Universal Robots URScript: external_control.urscript

{{BEGIN_REPLACE}}

# HEADER_BEGIN

steptime = get_steptime()

textmsg("ExternalControl: steptime=", steptime)
MULT_jointstate = {{JOINT_STATE_REPLACE}}
MULT_time = {{TIME_REPLACE}}

STOPJ_ACCELERATION = 4.0

#Constants
SERVO_UNINITIALIZED = -1
SERVO_IDLE = 0
SERVO_RUNNING = 1

MODE_STOPPED = -2
MODE_UNINITIALIZED = -1
MODE_IDLE = 0
MODE_SERVOJ = 1
MODE_SPEEDJ = 2
MODE_FORWARD = 3
MODE_SPEEDL = 4
MODE_POSE = 5
MODE_SPLINE = 6

TRAJECTORY_MODE_RECEIVE = 1
TRAJECTORY_MODE_CANCEL = -1

TRAJECTORY_POINT_INTERPOLATION = 0
TRAJECTORY_SPLINE_INTERPOLATION = 1

TRAJECTORY_POINT_JOINT = 0
TRAJECTORY_POINT_CARTESIAN = 1
TRAJECTORY_DATA_DIMENSION = 7

TRAJECTORY_RESULT_SUCCESS = 0
TRAJECTORY_RESULT_CANCELED = 1
TRAJECTORY_RESULT_FAILURE = 2

CUBIC_SPLINES = 0
QUINTIC_SPLINES = 1

TRAJECTORY_SPLINE_DATA_DIMENSION = 3*6 + 2

#Global variables are also showed in the Teach pendants variable list
global cmd_servo_state = SERVO_UNINITIALIZED
global cmd_servo_qd = [0.0, 0.0, 0.0, 0.0, 0.0, 0.0]
global cmd_servo_q = get_actual_joint_positions()
global cmd_servo_q_last = get_actual_joint_positions()
global cmd_twist = [0.0, 0.0, 0.0, 0.0, 0.0, 0.0]
global extrapolate_count = 0
global extrapolate_max_count = 0
global control_mode = MODE_UNINITIALIZED
global trajectory_points_left = 0

def set_servo_setpoint(params_mult):
  cmd_servo_state = SERVO_RUNNING
  cmd_servo_q_last = cmd_servo_q
  cmd_servo_q = [params_mult[2] / MULT_jointstate, params_mult[3] / MULT_jointstate, params_mult[4] / MULT_jointstate, params_mult[5] / MULT_jointstate, params_mult[6] / MULT_jointstate, params_mult[7] / MULT_jointstate]
end

def extrapolate():
  diff = [cmd_servo_q[0] - cmd_servo_q_last[0], cmd_servo_q[1] - cmd_servo_q_last[1], cmd_servo_q[2] - cmd_servo_q_last[2], cmd_servo_q[3] - cmd_servo_q_last[3], cmd_servo_q[4] - cmd_servo_q_last[4], cmd_servo_q[5] - cmd_servo_q_last[5]]
  cmd_servo_q_last = cmd_servo_q
  cmd_servo_q = [cmd_servo_q[0] + diff[0], cmd_servo_q[1] + diff[1], cmd_servo_q[2] + diff[2], cmd_servo_q[3] + diff[3], cmd_servo_q[4] + diff[4], cmd_servo_q[5] + diff[5]]

  return cmd_servo_q
end

thread servoThread():
  textmsg("ExternalControl: Starting servo thread")
  state = SERVO_IDLE
  while control_mode == MODE_SERVOJ:
    enter_critical
    q = cmd_servo_q
    do_extrapolate = False
    if (cmd_servo_state == SERVO_IDLE):
      do_extrapolate = True
    end
    state = cmd_servo_state
    if cmd_servo_state > SERVO_UNINITIALIZED:
      cmd_servo_state = SERVO_IDLE
    end

    if do_extrapolate:
      extrapolate_count = extrapolate_count + 1
      if extrapolate_count > extrapolate_max_count:
        extrapolate_max_count = extrapolate_count
      end

      q = extrapolate()
      servoj(q, t=steptime, {{SERVO_J_REPLACE}})

    elif state == SERVO_RUNNING:
      extrapolate_count = 0
      servoj(q, t=steptime, {{SERVO_J_REPLACE}})
    else:
      extrapolate_count = 0
      sync()
    end
    exit_critical
  end
  textmsg("ExternalControl: servo thread ended")
  stopj(STOPJ_ACCELERATION)
end

# Helpers for speed control
def set_speed(params_mult):
  cmd_servo_qd = [params_mult[2] / MULT_jointstate, params_mult[3] / MULT_jointstate, params_mult[4] / MULT_jointstate, params_mult[5] / MULT_jointstate, params_mult[6] / MULT_jointstate, params_mult[7] / MULT_jointstate]
  control_mode = MODE_SPEEDJ
end

thread speedThread():
  textmsg("ExternalControl: Starting speed thread")
  while control_mode == MODE_SPEEDJ:
    qd = cmd_servo_qd
    speedj(qd, 40.0, steptime)
  end
  textmsg("ExternalControl: speedj thread ended")
  stopj(STOPJ_ACCELERATION)
end

coefficients0 = [0.0, 0.0, 0.0, 0.0, 0.0, 0.0]
coefficients1 = [0.0, 0.0, 0.0, 0.0, 0.0, 0.0]
coefficients2 = [0.0, 0.0, 0.0, 0.0, 0.0, 0.0]
coefficients3 = [0.0, 0.0, 0.0, 0.0, 0.0, 0.0]
coefficients4 = [0.0, 0.0, 0.0, 0.0, 0.0, 0.0]
coefficients5 = [0.0, 0.0, 0.0, 0.0, 0.0, 0.0]
cartesian_coefficients0 = [0.0, 0.0, 0.0, 0.0, 0.0, 0.0, 0.0]
cartesian_coefficients1 = [0.0, 0.0, 0.0, 0.0, 0.0, 0.0, 0.0]
cartesian_coefficients2 = [0.0, 0.0, 0.0, 0.0, 0.0, 0.0, 0.0]
cartesian_coefficients3 = [0.0, 0.0, 0.0, 0.0, 0.0, 0.0, 0.0]
cartesian_coefficients4 = [0.0, 0.0, 0.0, 0.0, 0.0, 0.0, 0.0]
cartesian_coefficients5 = [0.0, 0.0, 0.0, 0.0, 0.0, 0.0, 0.0]
splineTimer = 0.0
splineTravelTime = 0.0

def reset_spline_coefficents():
  coefficients0 = [0.0, 0.0, 0.0, 0.0, 0.0, 0.0]
  coefficients1 = [0.0, 0.0, 0.0, 0.0, 0.0, 0.0]
  coefficients2 = [0.0, 0.0, 0.0, 0.0, 0.0, 0.0]
  coefficients3 = [0.0, 0.0, 0.0, 0.0, 0.0, 0.0]
  coefficients4 = [0.0, 0.0, 0.0, 0.0, 0.0, 0.0]
  coefficients5 = [0.0, 0.0, 0.0, 0.0, 0.0, 0.0]

  cartesian_coefficients0 = [0.0, 0.0, 0.0, 0.0, 0.0, 0.0, 0.0]
  cartesian_coefficients1 = [0.0, 0.0, 0.0, 0.0, 0.0, 0.0, 0.0]
  cartesian_coefficients2 = [0.0, 0.0, 0.0, 0.0, 0.0, 0.0, 0.0]
  cartesian_coefficients3 = [0.0, 0.0, 0.0, 0.0, 0.0, 0.0, 0.0]
  cartesian_coefficients4 = [0.0, 0.0, 0.0, 0.0, 0.0, 0.0, 0.0]
  cartesian_coefficients5 = [0.0, 0.0, 0.0, 0.0, 0.0, 0.0, 0.0]

  splineTimer = 0.0
  splineTravelTime = 0.0
end

def cubic_spline_calculation(start_pos, end_pos, start_vel, end_vel, time):
  if time == 0.0:
    coefficients0 = start_pos
    coefficients1 = start_vel
    coefficients2 = coefficients2 * 0.0
    coefficients3 = coefficients3 * 0.0
  else:
    coefficients0 = start_pos
    coefficients1 = start_vel
    coefficients2 = (-3 * start_pos + end_pos * 3 - start_vel * 2 * time - end_vel * time) / pow(time,2)
    coefficients3 = (2 * start_pos - 2 * end_pos + start_vel * time + end_vel * time) / pow(time,3)
  end
  coefficients4 = coefficients4 * 0.0
  coefficients5 = coefficients5 * 0.0
  splineTimer = 0.0
  splineTravelTime = time
end

def quintic_spline_calculation(start_pos, end_pos, start_vel, end_vel, start_acc, end_acc, time):
  TIME1 =  time
  TIME2 = pow(time,2)
  TIME3 = pow(time,3)
  TIME4 = pow(time,4)
  TIME5 = pow(time,5)

  if time == 0.0:
    coefficients0 = start_pos
    coefficients1 = start_vel
    coefficients2 = 0.5*start_acc
    coefficients3 = coefficients3 * 0.0
    coefficients4 = coefficients4 * 0.0
    coefficients5 = coefficients5 * 0.0
  else:
    coefficients0 = start_pos
    coefficients1 = start_vel
    coefficients2 = 0.5*start_acc
    coefficients3 = (-20.0 * start_pos + 20.0 * end_pos - 3.0 * start_acc * TIME2 + end_acc * TIME2 - 12.0 * start_vel * time - 8.0 * end_vel * time) / (2.0 * TIME3)
    coefficients4 = (30.0 * start_pos - 30.0 * end_pos + 3.0* start_acc * TIME2 - 2.0 * end_acc * TIME2 + 16.0 * start_vel * time + 14.0 * end_vel * time) / (2.0 * TIME4)
    coefficients5 = (-12.0 * start_pos + 12.0 * end_pos - start_acc * TIME2 + end_acc * TIME2 - 6.0 * start_vel * time - 6.0 * end_vel * time) / (2.0 * TIME5)
  end
  splineTimer = 0.0
  splineTravelTime  = time
end

def joint_spline_run():
  spline_step_time = get_steptime()
  if splineTravelTime < spline_step_time:
    TIME1 = splineTimer
    TIME2  = pow(TIME1,2)
    TIME3  = pow(TIME1,3)
    TIME4  = pow(TIME1,4)
    qd = coefficients1 + 2.0*TIME1*coefficients2 + 3.0*TIME2*coefficients3 + 4.0*TIME3*coefficients4 + 5.0*TIME4*coefficients5
    speedj(qd,1000,spline_step_time)
  end

  splineTimer = splineTimer + spline_step_time
  while splineTimer <= splineTravelTime:
    TIME1 = splineTimer
    TIME2  = pow(TIME1,2)
    TIME3  = pow(TIME1,3)
    TIME4  = pow(TIME1,4)

    #q = coefficients0 + coefficients1 + TIME2*coefficients2 + TIME3*coefficients3 + TIME4*coefficients4 + TIME5*coefficients5
    qd = coefficients1 + 2.0*TIME1*coefficients2 + 3.0*TIME2*coefficients3 + 4.0*TIME3*coefficients4 + 5.0*TIME4*coefficients5

    speedj(qd,1000,spline_step_time)

    splineTimer = splineTimer + spline_step_time
  end
end

# Quaterion operations, the quaternion is expected to be an array of order [w, x, y, z]
def check_quaternion_length(q):
  if length(q) != 4:
    popup("Quaternion should have length 4", title="Quaternion has wrong length", error=True)
    halt
  end
end

def get_quaternion_conjugate(q):
  check_quaternion_length(q)
  return [q[0], -q[1], -q[2], -q[3]]
end

def get_quaternion_norm(q):
  check_quaternion_length(q)
  return sqrt(pow(q[0],2) + pow(q[1],2) + pow(q[2],2) + pow(q[3],2))
end

def normalize_quaternion(q):
  check_quaternion_length(q)
  return q / get_quaternion_norm(q)
end

def get_inverse_quaternion(q):
  check_quaternion_length(q)
  return get_quaternion_conjugate(q) / pow(get_quaternion_norm(q),2)
end

def quaternion_multiplication(a, b):
  check_quaternion_length(a)
  check_quaternion_length(b)
  q = [a[0]*b[0] - a[1]*b[1] - a[2]*b[2] - a[3]*b[3],
       a[0]*b[1] + a[1]*b[0] + a[2]*b[3] - a[3]*b[2],
       a[0]*b[2] + a[2]*b[0] + a[3]*b[1] - a[1]*b[3],
       a[0]*b[3] + a[3]*b[0] + a[1]*b[2] - a[2]*b[1]]
  return q
end

def quaternion_to_axis_angle(q):
  check_quaternion_length(q)
  q_normalized = normalize_quaternion(q)
  angle = 2 * atan2(norm([q_normalized[1], q_normalized[2], q_normalized[3]]), q_normalized[0])
  axis = [q_normalized[1], q_normalized[2], q_normalized[3]]
  if norm(angle) > 0.001:
    axis = axis / sin(angle/2)
  end
  return angle * axis
end

def axis_angle_to_quaternion(aa):
  if length(aa) != 3:
    popup("Angle axis should have length 3", title="Angle axis has wrong length", error=True)
    halt
  end
  angle = norm(aa)
  if (norm(angle) < 10e-7):
    axis = [0, 0, 0]
    anlge = 0
  else:
    axis = (aa / angle) * sin(angle/2)
  end
  return [cos(angle/2), axis[0], axis[1], axis[2]]
end

# Converts the cartesian state into a spline state, so that the trajectory can be interpolated
# This is based on the math from
# https://github.com/UniversalRobots/Universal_Robots_ROS_controllers_cartesian/blob/main/cartesian_trajectory_interpolation/include/cartesian_trajectory_interpolation/cartesian_trajectory_segment.h
def convert_to_spline_state(pose, vel, acc=[]):
  q = normalize_quaternion([pose[3], pose[4], pose[5], pose[6]])
  inverse_q = get_inverse_quaternion(q)

  # transform rotational velocities into body local reference frame
  omega = quaternion_multiplication(inverse_q, [0, vel[3], vel[4], vel[5]])
  omega = quaternion_multiplication(omega, q)
  omega[0] = 0
  q_dot = 0.5 * quaternion_multiplication(q, omega)

  # transform positional velocities into body local reference frame
  x_dot = quaternion_multiplication(inverse_q, [0, vel[0], vel[1], vel[2]])
  x_dot = quaternion_multiplication(x_dot, q)

  if size(acc) == 0:
    # Create spline state vector
    spline_state = [pose[0], pose[1], pose[2], q[0], q[1], q[2], q[3],
                    x_dot[1], x_dot[2], x_dot[3], q_dot[0], q_dot[1], q_dot[2], q_dot[3]]

    return spline_state
  end

  # transform rotational acceleration into body local reference frame
  omega_dot = quaternion_multiplication(inverse_q, [0, acc[3], acc[4], acc[5]])
  omega_dot = quaternion_multiplication(omega_dot, q)
  omega_dot[0] = 0
  q_ddot = 0.5 * quaternion_multiplication(q, omega_dot) + 0.5 * quaternion_multiplication(q_dot, omega)

  # transform positional acceleration into body local reference frame
  x_ddot = quaternion_multiplication(inverse_q, [0, acc[0], acc[1], acc[2]])
  x_ddot = quaternion_multiplication(x_ddot, q)

  # Create spline state
  spline_state = [pose[0], pose[1], pose[2], q[0], q[1], q[2], q[3],
                  x_dot[1], x_dot[2], x_dot[3], q_dot[0], q_dot[1], q_dot[2], q_dot[3],
                  x_ddot[1], x_ddot[2], x_ddot[3], q_ddot[0], q_ddot[1], q_ddot[2], q_ddot[3]]

  return spline_state
end

# Converts the spline state back into cartesian state
# This is based on the math from
# https://github.com/UniversalRobots/Universal_Robots_ROS_controllers_cartesian/blob/main/cartesian_trajectory_interpolation/include/cartesian_trajectory_interpolation/cartesian_trajectory_segment.h
def convert_to_cartesian_state(pos, vel):
  q = normalize_quaternion([pos[3], pos[4], pos[5], pos[6]])
  inverse_q = get_inverse_quaternion(q)

  omega = 2.0 * quaternion_multiplication(inverse_q, [vel[3], vel[4], vel[5], vel[6]])
  omega[0] = 0
  omega = quaternion_multiplication(q, omega)
  omega = quaternion_multiplication(omega, inverse_q)

  x_dot = quaternion_multiplication(q, [0, vel[0], vel[1], vel[2]])
  x_dot = quaternion_multiplication(x_dot, inverse_q)

  twist = [x_dot[1], x_dot[2], x_dot[3], omega[1], omega[2], omega[3]]
  return twist
end

def cubic_cartesian_spline_calculation(start_position, end_position, start_velocity, end_velocity, time):
  # If the dot product is negative, we change the sing of the orientation to not travel the long way around
  dot_product = start_position[3]*end_position[3] + start_position[4]*end_position[4] + start_position[5]*end_position[5] + start_position[6]*end_position[6]
  if dot_product < 0.0:
    end_position[3] = end_position[3] * - 1
    end_position[4] = end_position[4] * - 1
    end_position[5] = end_position[5] * - 1
    end_position[6] = end_position[6] * - 1
  end

  start_state = convert_to_spline_state(start_position, start_velocity)
  end_state = convert_to_spline_state(end_position, end_velocity)

  # Get position
  start_pos = [start_state[0], start_state[1], start_state[2], start_state[3],
                start_state[4], start_state[5], start_state[6]]
  end_pos = [end_state[0], end_state[1], end_state[2], end_state[3],
                end_state[4], end_state[5], end_state[6]]

  # Get velocity
  start_vel = [start_state[7], start_state[8], start_state[9], start_state[10],
                start_state[11], start_state[12], start_state[13]]
  end_vel = [end_state[7], end_state[8], end_state[9], end_state[10],
                end_state[11], end_state[12], end_state[13]]

  if time == 0.0:
    cartesian_coefficients0 = start_pos
    cartesian_coefficients1 = start_vel
    cartesian_coefficients2 = cartesian_coefficients2 * 0.0
    cartesian_coefficients3 = cartesian_coefficients3 * 0.0
  else:
    cartesian_coefficients0 = start_pos
    cartesian_coefficients1 = start_vel
    cartesian_coefficients2 = (-3 * start_pos + end_pos * 3 - start_vel * 2 * time - end_vel * time) / pow(time,2)
    cartesian_coefficients3 = (2 * start_pos - 2 * end_pos + start_vel * time + end_vel * time) / pow(time,3)
  end
  cartesian_coefficients4 = cartesian_coefficients4 * 0.0
  cartesian_coefficients5 = cartesian_coefficients5 * 0.0
  splineTimer = 0.0
  splineTravelTime = time
end

def quintic_cartesian_spline_calculation(start_position, end_position, start_velocity, end_velocity, start_acceleration, end_acceleration, time):
  # If the dot product is negative, we change the sing of the orientation to not travel the long way around
  dot_product = start_position[3]*end_position[3] + start_position[4]*end_position[4] + start_position[5]*end_position[5] + start_position[6]*end_position[6]
  if dot_product < 0.0:
    end_position[3] = end_position[3] * - 1
    end_position[4] = end_position[4] * - 1
    end_position[5] = end_position[5] * - 1
    end_position[6] = end_position[6] * - 1
  end

  start_spline_state = convert_to_spline_state(start_position, start_velocity, start_acceleration)
  end_spline_state = convert_to_spline_state(end_position, end_velocity, end_acceleration)

  # Get position
  start_pos = [start_spline_state[0], start_spline_state[1], start_spline_state[2], start_spline_state[3],
                start_spline_state[4], start_spline_state[5], start_spline_state[6]]
  end_pos = [end_spline_state[0], end_spline_state[1], end_spline_state[2], end_spline_state[3],
              end_spline_state[4], end_spline_state[5], end_spline_state[6]]

  # Get velocity
  start_vel = [start_spline_state[7], start_spline_state[8], start_spline_state[9], start_spline_state[10],
               start_spline_state[11], start_spline_state[12], start_spline_state[13]]
  end_vel = [end_spline_state[7], end_spline_state[8], end_spline_state[9], end_spline_state[10],
             end_spline_state[11], end_spline_state[12], end_spline_state[13]]

  # Get Acceleration
  start_acc = [start_spline_state[14], start_spline_state[15], start_spline_state[16], start_spline_state[17],
               start_spline_state[18], start_spline_state[19], start_spline_state[20]]
  end_acc = [end_spline_state[14], end_spline_state[15], end_spline_state[16], end_spline_state[17],
             end_spline_state[18], end_spline_state[19], end_spline_state[20]]

  TIME1 =  time
  TIME2 = pow(time,2)
  TIME3 = pow(time,3)
  TIME4 = pow(time,4)
  TIME5 = pow(time,5)

  if time == 0.0:
    cartesian_coefficients0 = start_pos
    cartesian_coefficients1 = start_vel
    cartesian_coefficients2 = 0.5*start_acc
    cartesian_coefficients3 = cartesian_coefficients3 * 0.0
    cartesian_coefficients4 = cartesian_coefficients4 * 0.0
    cartesian_coefficients5 = cartesian_coefficients5 * 0.0
  else:
    cartesian_coefficients0 = start_pos
    cartesian_coefficients1 = start_vel
    cartesian_coefficients2 = 0.5*start_acc
    cartesian_coefficients3 = (-20.0 * start_pos + 20.0 * end_pos - 3.0 * start_acc * TIME2 + end_acc * TIME2 - 12.0 * start_vel * time - 8.0 * end_vel * time) / (2.0 * TIME3)
    cartesian_coefficients4 = (30.0 * start_pos - 30.0 * end_pos + 3.0* start_acc * TIME2 - 2.0 * end_acc * TIME2 + 16.0 * start_vel * time + 14.0 * end_vel * time) / (2.0 * TIME4)
    cartesian_coefficients5 = (-12.0 * start_pos + 12.0 * end_pos - start_acc * TIME2 + end_acc * TIME2 - 6.0 * start_vel * time - 6.0 * end_vel * time) / (2.0 * TIME5)
  end
  splineTimer = 0.0
  splineTravelTime  = time
end

def cartesian_spline_run():
  spline_step_time = get_steptime()
  if splineTravelTime < spline_step_time:
    TIME1 = splineTimer
    TIME2  = pow(TIME1,2)
    TIME3  = pow(TIME1,3)
    TIME4  = pow(TIME1,4)
    TIME5  = pow(TIME1,5)
    pose = cartesian_coefficients0 + TIME1*cartesian_coefficients1 + TIME2*cartesian_coefficients2 + TIME3*cartesian_coefficients3 + TIME4*cartesian_coefficients4 + TIME5*cartesian_coefficients5
    vel = cartesian_coefficients1 + 2.0*TIME1*cartesian_coefficients2 + 3.0*TIME2*cartesian_coefficients3 + 4.0*TIME3*cartesian_coefficients4 + 5.0*TIME4*cartesian_coefficients5
    twist = convert_to_cartesian_state(pose, vel)
    speedl(twist,1000,spline_step_time)
  end

  splineTimer = splineTimer + spline_step_time
  while splineTimer <= splineTravelTime:
    TIME1 = splineTimer
    TIME2  = pow(TIME1,2)
    TIME3  = pow(TIME1,3)
    TIME4  = pow(TIME1,4)
    TIME5  = pow(TIME1,5)
    pose = cartesian_coefficients0 + TIME1*cartesian_coefficients1 + TIME2*cartesian_coefficients2 + TIME3*cartesian_coefficients3 + TIME4*cartesian_coefficients4 + TIME5*cartesian_coefficients5
    vel = cartesian_coefficients1 + 2.0*TIME1*cartesian_coefficients2 + 3.0*TIME2*cartesian_coefficients3 + 4.0*TIME3*cartesian_coefficients4 + 5.0*TIME4*cartesian_coefficients5
    aa = quaternion_to_axis_angle([pose[3], pose[4], pose[5], pose[6]])
    cmd_servo_q = get_inverse_kin(p[pose[0], pose[1], pose[2], aa[0], aa[1], aa[2]], get_actual_joint_positions())
    #twist = convert_to_cartesian_state(pose, vel)
    #speedl(twist,1000,spline_step_time)
    servoj(cmd_servo_q, t=spline_step_time, {{SERVO_J_REPLACE}})
    splineTimer = splineTimer + spline_step_time
  end
end

thread jointTrajectoryThread():
  textmsg("Executing trajectory. Number of points: ", trajectory_points_left)
  local INDEX_TIME = TRAJECTORY_DATA_DIMENSION
  local INDEX_BLEND = INDEX_TIME + 1
  local INDEX_POINT_TYPE = INDEX_BLEND + 1
  while trajectory_points_left > 0:
    enter_critical
    #reading trajectory point + blend radius + type of point (cartesian/joint based)
    raw_point = socket_read_binary_integer(TRAJECTORY_DATA_DIMENSION+1+1, "trajectory_socket")
    trajectory_points_left = trajectory_points_left - 1
    exit_critical
    if raw_point[0] > 0:
      q = [ raw_point[1] / MULT_jointstate, raw_point[2] / MULT_jointstate, raw_point[3] / MULT_jointstate, raw_point[4] / MULT_jointstate, raw_point[5] / MULT_jointstate, raw_point[6] / MULT_jointstate]
      tmptime = raw_point[INDEX_TIME] / MULT_time
      blend_radius = raw_point[INDEX_BLEND] / MULT_time

      if trajectory_points_left > 0:
        if raw_point[INDEX_POINT_TYPE] == TRAJECTORY_POINT_JOINT:
          # textmsg("Executing movej with blending")
          movej(q, t=tmptime, r=blend_radius)
        elif raw_point[INDEX_POINT_TYPE] == TRAJECTORY_POINT_CARTESIAN:
          # textmsg("Executing movel with blending")
          movel(p[q[0], q[1], q[2], q[3], q[4], q[5]], t=tmptime, r=blend_radius)
        end
      else:
        if raw_point[INDEX_POINT_TYPE] == TRAJECTORY_POINT_JOINT:
          # textmsg("Executing movej without blending")
          movej(q, t=tmptime, r=0.0)
        elif raw_point[INDEX_POINT_TYPE] == TRAJECTORY_POINT_CARTESIAN:
          # textmsg("Executing movel without blending")
          movel(p[q[0], q[1], q[2], q[3], q[4], q[5]], t=tmptime, r=0.0)
        end
      end
    end
  end
  socket_send_int(TRAJECTORY_RESULT_SUCCESS, "trajectory_socket")
  textmsg("Trajectory finished")
end

# Helper functions
def get_tcp_position_as_list():
  actual_tcp_pose = get_actual_tcp_pose()
  q = axis_angle_to_quaternion([actual_tcp_pose[3], actual_tcp_pose[4], actual_tcp_pose[5]])
  return [actual_tcp_pose[0], actual_tcp_pose[1], actual_tcp_pose[2], q[0], q[1], q[2], q[3]]
end

def get_tcp_speed_as_list():
  actual_tcp_speed = get_actual_tcp_speed()
  return [actual_tcp_speed[0], actual_tcp_speed[1], actual_tcp_speed[2], actual_tcp_speed[3], actual_tcp_speed[4], actual_tcp_speed[4]]
end

thread splineThread():
  textmsg("Executing trajectory. Number of points: ", trajectory_points_left)
  local INDEX_TIME = TRAJECTORY_SPLINE_DATA_DIMENSION
  local INDEX_SPLINE_TYPE = INDEX_TIME + 1
  local INDEX_POINT_TYPE = INDEX_SPLINE_TYPE + 1
  old_qdd = [0, 0, 0, 0, 0, 0]
  old_cart_acc = [0, 0, 0, 0, 0, 0]
  reset_spline_coefficents()
  while trajectory_points_left > 0:
    # reading trajectory point + spline type
    enter_critical
    raw_point = socket_read_binary_integer(TRAJECTORY_SPLINE_DATA_DIMENSION+2, "trajectory_socket")
    trajectory_points_left = trajectory_points_left - 1
    exit_critical
    if raw_point[0] > 0:
      tmptime = raw_point[INDEX_TIME] / MULT_time
      if trajectory_points_left > 0:
        textmsg("point type ", raw_point[INDEX_SPLINE_TYPE])
        if raw_point[INDEX_POINT_TYPE] == TRAJECTORY_POINT_CARTESIAN:
          cart_pos = [ raw_point[1] / MULT_jointstate, raw_point[2] / MULT_jointstate, raw_point[3] / MULT_jointstate, raw_point[4] / MULT_jointstate, raw_point[5] / MULT_jointstate, raw_point[6] / MULT_jointstate, raw_point[7] / MULT_jointstate]
          cart_vel = [ raw_point[8] / MULT_jointstate, raw_point[9] / MULT_jointstate, raw_point[10] / MULT_jointstate, raw_point[11] / MULT_jointstate, raw_point[12] / MULT_jointstate, raw_point[13] / MULT_jointstate]
          if raw_point[INDEX_SPLINE_TYPE] == CUBIC_SPLINES:
            cubic_cartesian_spline_calculation(get_tcp_position_as_list(), cart_pos, get_tcp_speed_as_list(), cart_vel, tmptime)
            old_cart_acc = [0, 0, 0, 0, 0, 0, 0]
          elif raw_point[INDEX_SPLINE_TYPE] == QUINTIC_SPLINES:
            cart_acc = [ raw_point[14] / MULT_jointstate, raw_point[15] / MULT_jointstate, raw_point[16] / MULT_jointstate, raw_point[17] / MULT_jointstate, raw_point[18] / MULT_jointstate, raw_point[19] / MULT_jointstate]
            cubic_cartesian_spline_calculation(get_tcp_position_as_list(), cart_pos, get_tcp_speed_as_list(), cart_vel, tmptime)
            old_cart_acc = cart_acc
          end
          cartesian_spline_run()
        elif raw_point[INDEX_POINT_TYPE] == TRAJECTORY_POINT_JOINT:
          q = [ raw_point[1] / MULT_jointstate, raw_point[2] / MULT_jointstate, raw_point[3] / MULT_jointstate, raw_point[4] / MULT_jointstate, raw_point[5] / MULT_jointstate, raw_point[6] / MULT_jointstate]
          qd = [ raw_point[8] / MULT_jointstate, raw_point[9] / MULT_jointstate, raw_point[10] / MULT_jointstate, raw_point[11] / MULT_jointstate, raw_point[12] / MULT_jointstate, raw_point[13] / MULT_jointstate]
          if raw_point[INDEX_SPLINE_TYPE] == CUBIC_SPLINES:
            cubic_spline_calculation(get_actual_joint_positions(), q, get_actual_joint_speeds(), qd, tmptime)
            old_qdd = [0, 0, 0, 0, 0, 0]
          elif raw_point[INDEX_SPLINE_TYPE] == QUINTIC_SPLINES:
            qdd = [ raw_point[14] / MULT_jointstate, raw_point[15] / MULT_jointstate, raw_point[16] / MULT_jointstate, raw_point[17] / MULT_jointstate, raw_point[18] / MULT_jointstate, raw_point[19] / MULT_jointstate]
            quintic_spline_calculation(get_actual_joint_positions(),q, get_actual_joint_speeds(), qd, old_qdd, qdd, tmptime)
            old_qdd = qdd
          end
          joint_spline_run()
        end
      else:
        if raw_point[INDEX_POINT_TYPE] == TRAJECTORY_POINT_CARTESIAN:
          cart_pos = [ raw_point[1] / MULT_jointstate, raw_point[2] / MULT_jointstate, raw_point[3] / MULT_jointstate, raw_point[4] / MULT_jointstate, raw_point[5] / MULT_jointstate, raw_point[6] / MULT_jointstate, raw_point[7] / MULT_jointstate]
          cubic_cartesian_spline_calculation(get_tcp_position_as_list(), cart_pos, get_tcp_speed_as_list(), [0,0,0,0,0,0], tmptime)
          cartesian_spline_run()
        elif raw_point[INDEX_POINT_TYPE] == TRAJECTORY_POINT_JOINT:
          q = [ raw_point[1] / MULT_jointstate, raw_point[2] / MULT_jointstate, raw_point[3] / MULT_jointstate, raw_point[4] / MULT_jointstate, raw_point[5] / MULT_jointstate, raw_point[6] / MULT_jointstate]
          qd = [ raw_point[8] / MULT_jointstate, raw_point[9] / MULT_jointstate, raw_point[10] / MULT_jointstate, raw_point[11] / MULT_jointstate, raw_point[12] / MULT_jointstate, raw_point[13] / MULT_jointstate]
          cubic_spline_calculation(get_actual_joint_positions(), q, get_actual_joint_speeds(), [0,0,0,0,0,0], tmptime)
          joint_spline_run()
        end
      end
    end
  end
  socket_send_int(TRAJECTORY_RESULT_SUCCESS, "trajectory_socket")
  textmsg("Trajectory finished")
end

def clear_remaining_trajectory_points():
  while trajectory_points_left > 0:
    raw_point = socket_read_binary_integer(TRAJECTORY_DATA_DIMENSION+2, "trajectory_socket")
    trajectory_points_left = trajectory_points_left - 1
  end
  reset_spline_coefficents()
end

# Helpers for speed control
def set_speedl(params_mult):
  cmd_twist = [params_mult[2] / MULT_jointstate, params_mult[3] / MULT_jointstate, params_mult[4] / MULT_jointstate, params_mult[5] / MULT_jointstate, params_mult[6] / MULT_jointstate, params_mult[7] / MULT_jointstate]
  control_mode = MODE_SPEEDL
end

thread speedlThread():
  textmsg("Starting speedl thread")
  while control_mode == MODE_SPEEDL:
    twist = cmd_twist
    speedl(twist, 40.0, steptime)
  end
  textmsg("speedl thread ended")
  stopj(STOPJ_ACCELERATION)
end

thread servoThreadP():
  textmsg("Starting pose servo thread")
  state = SERVO_IDLE
  while control_mode == MODE_POSE:
    enter_critical
    q = cmd_servo_q
    do_extrapolate = False
    if (cmd_servo_state == SERVO_IDLE):
      do_extrapolate = True
    end
    state = cmd_servo_state
    if cmd_servo_state > SERVO_UNINITIALIZED:
      cmd_servo_state = SERVO_IDLE
    end

    if do_extrapolate:
      extrapolate_count = extrapolate_count + 1
      if extrapolate_count > extrapolate_max_count:
        extrapolate_max_count = extrapolate_count
      end

      q = extrapolate()
      servoj(q, t=steptime, {{SERVO_J_REPLACE}})

    elif state == SERVO_RUNNING:
      extrapolate_count = 0
      servoj(q, t=steptime, {{SERVO_J_REPLACE}})
    else:
      extrapolate_count = 0
      sync()
    end
    exit_critical
  end
  textmsg("pose servo thread ended")
  stopj(STOPJ_ACCELERATION)
end

def set_servo_pose(params_mult):
  pose = p[params_mult[2] / MULT_jointstate, params_mult[3] / MULT_jointstate, params_mult[4] / MULT_jointstate, params_mult[5] / MULT_jointstate, params_mult[6] / MULT_jointstate, params_mult[7] / MULT_jointstate]
  cmd_servo_state = SERVO_RUNNING
  cmd_servo_q_last = cmd_servo_q
  cmd_servo_q = get_inverse_kin(pose, cmd_servo_q)
end


# HEADER_END

# NODE_CONTROL_LOOP_BEGINS

socket_open("{{SERVER_IP_REPLACE}}", {{SERVER_PORT_REPLACE}}, "reverse_socket")
socket_open("{{SERVER_IP_REPLACE}}", {{TRAJECTORY_SERVER_PORT_REPLACE}}, "trajectory_socket")

control_mode = MODE_UNINITIALIZED
thread_move = 0
thread_trajectory = 0
trajectory_points_left = 0
global keepalive = -2
read_timeout = 0.02
params_mult = socket_read_binary_integer(1+6+1, "reverse_socket", 0)
textmsg("ExternalControl: External control active")
keepalive = params_mult[1]
while keepalive > 0 and control_mode > MODE_STOPPED:
  enter_critical
  params_mult = socket_read_binary_integer(1+6+1, "reverse_socket", read_timeout)
  if params_mult[0] > 0:
    keepalive = params_mult[1]

    # New control mode received
    if control_mode != params_mult[8]:
      #Stop the trajectory and flush the point in pipeline
      if control_mode == MODE_FORWARD:
        kill thread_trajectory
        stopj(STOPJ_ACCELERATION)
        clear_remaining_trajectory_points()
      else:
        kill thread_move
        stopj(STOPJ_ACCELERATION)
      end


      #Run the new type of motion
      control_mode = params_mult[8]
      if control_mode == MODE_SERVOJ:
        thread_move = run servoThread()
      elif control_mode == MODE_SPEEDJ:
        thread_move = run speedThread()
      elif control_mode == MODE_FORWARD:
        kill thread_move
      elif control_mode == MODE_SPEEDL:
        thread_move = run speedlThread()
      elif control_mode == MODE_POSE:
        thread_move = run servoThreadP()
      end
    end

    # Update the motion commands with new parameters
    if control_mode == MODE_SERVOJ:
      set_servo_setpoint(params_mult)
    elif control_mode == MODE_SPEEDJ:
      set_speed(params_mult)
    elif control_mode == MODE_FORWARD:
      if params_mult[2] == TRAJECTORY_MODE_RECEIVE:
        kill thread_trajectory
        clear_remaining_trajectory_points()
        trajectory_points_left = params_mult[3]
        if TRAJECTORY_POINT_INTERPOLATION == params_mult[4]:
          thread_trajectory = run jointTrajectoryThread()
        elif TRAJECTORY_SPLINE_INTERPOLATION == params_mult[4]:
          thread_trajectory = run splineThread()
        end
      elif params_mult[2] == TRAJECTORY_MODE_CANCEL:
        textmsg("cancel received")
        kill thread_trajectory
        clear_remaining_trajectory_points()
        socket_send_int(TRAJECTORY_RESULT_CANCELED, "trajectory_socket")
      end
    elif control_mode == MODE_SPEEDL:
      set_speedl(params_mult)
    elif control_mode == MODE_POSE:
      set_servo_pose(params_mult)
    end
  else:
    keepalive = keepalive - 1
  end
  exit_critical
end

textmsg("ExternalControl: Stopping communication and control")
control_mode = MODE_STOPPED
join thread_move
join thread_trajectory
textmsg("ExternalControl: All threads ended")
socket_close("reverse_socket")
socket_close("trajectory_socket")

# NODE_CONTROL_LOOP_ENDS
